PROGRAM INTERNAL PRG_TEST_CONVERSION
VAR
 	bEnableTests : BOOL;

	in_dt : DATE_AND_TIME;
	out_str : STRING;
END_VAR

IF bEnableTests THEN
	out_str := Dt_To_Str(in_dt);
END_IF

END_PROGRAM

(* stored: Version 1.1.0.1, ProductVersion 3.1.4024.11
   POU PRG_TEST_CONVERSION: Id {6d253267-c11b-0916-38f7-c1d63cc7dc12}, SpecialFunc None *)
